(* IEC 61131-3 sources: programs/VI-54/VI-54_20171205/VI-54_20171205/Stations/Screen/LseClass170718/Class/SleegersControl, 1 file *)

(* ---- SleegersControl.st ---- *)
(*!
<Class
	Name               = "SleegersControl"
	Revision           = "0.0"
	RealtimeTask       = "false"
	CyclicTask         = "true"
	BackgroundTask     = "false"
	Sigmatek           = "false"
	OSInterface        = "false"
	HighPriority       = "false"
	Automatic          = "false"
	UpdateMode         = "Prescan"
	SharedCommandTable = "true"
	Objectsize         = "(570,120)">
	<Channels>
		<Server Name="BackToOldScreen" Visualized="true" Initialize="false" WriteProtected="false" Retentive="false"/>
		<Server Name="CarButtonHw" Visualized="true" Initialize="false" WriteProtected="true" Retentive="false"/>
		<Server Name="CarRecipes" Visualized="true" Initialize="false" WriteProtected="false" Retentive="false"/>
		<Server Name="ClassSvr" Visualized="false" Initialize="false" WriteProtected="true" Retentive="false"/>
		<Server Name="Index" Visualized="true" Initialize="false" WriteProtected="false" Retentive="false"/>
		<Server Name="OffsetCaroucelHw" Visualized="true" Initialize="false" WriteProtected="false" Retentive="false"/>
		<Server Name="ScrollBar" Visualized="true" Initialize="false" WriteProtected="false" Retentive="false"/>
		<Client Name="coAccessControlMain" Required="true" Internal="false"/>
		<Client Name="CommTerminal" Required="true" Internal="false"/>
		<Client Name="NewScreen" Required="true" Internal="false"/>
	</Channels>
</Class>
*)
SleegersControl : CLASS
  //Servers:
	ClassSvr 	: SvrChCmd_DINT;
	OffsetCaroucelHw 	: SvrCh_DINT;
	CarButtonHw 	: SvrCh_DINT;
	CarRecipes 	: SvrCh_DINT;
	Index 	: SvrCh_DINT;
	BackToOldScreen 	: SvrCh_DINT;
	ScrollBar 	: SvrCh_DINT;
  //Clients:
	coAccessControlMain 	: CltChCmd_AccessControlMain;
	NewScreen 	: CltCh_DINT;
	CommTerminal 	: CltChCmd_TerminalControl;
  //Variables:
		OldScreenNbr 	: DINT;
		Offset 	: DINT;
		OldScreen 	: DINT;
		ActScreen 	: DINT;
  //Functions:

	FUNCTION VIRTUAL GLOBAL Init;

	FUNCTION VIRTUAL GLOBAL CyWork
		VAR_INPUT
			EAX 	: UDINT;
		END_VAR
		VAR_OUTPUT
			state (EAX) 	: UDINT;
		END_VAR;

	FUNCTION GLOBAL OpenScreenAfterUnlock;

	FUNCTION VIRTUAL GLOBAL OffsetCaroucelHw::Write
		VAR_INPUT
			input (EAX) 	: DINT;
		END_VAR
		VAR_OUTPUT
			result (EAX) 	: DINT;
		END_VAR;

	FUNCTION VIRTUAL GLOBAL CarRecipes::Write
		VAR_INPUT
			input (EAX) 	: DINT;
		END_VAR
		VAR_OUTPUT
			result (EAX) 	: DINT;
		END_VAR;

	FUNCTION VIRTUAL GLOBAL Index::Write
		VAR_INPUT
			input (EAX) 	: DINT;
		END_VAR
		VAR_OUTPUT
			result (EAX) 	: DINT;
		END_VAR;

	FUNCTION VIRTUAL GLOBAL BackToOldScreen::Write
		VAR_INPUT
			input (EAX) 	: DINT;
		END_VAR
		VAR_OUTPUT
			result (EAX) 	: DINT;
		END_VAR;
  //Tables:
	FUNCTION @STD
		VAR_OUTPUT
			ret_code	: CONFSTATES;
		END_VAR;
	FUNCTION GLOBAL TAB @CT_;
END_CLASS;

#pragma usingLtd AccessControlMain
#pragma usingLtd TerminalControl

FUNCTION VIRTUAL GLOBAL SleegersControl::Init

  // Set actScreen
  ActScreen := CommTerminal.ActScreenNbr;

 // Set carroucel te one
 CarButtonHw := 1;

 // define screen numbers
 #define SMainHardware 7

 #define SVI46 48
 #define SVI11 49
 #define SVI47 50
 #define SVI48 51
 #define SVI49 52
 #define SVI50 53

 #define Salarm 22

 // define carroucel distances (offsets)
 #define OHardwareCards 550
 #define OMainHardware 600
 #define OAlarm 829

END_FUNCTION

FUNCTION VIRTUAL GLOBAL SleegersControl::CyWork
	VAR_INPUT
		EAX 	: UDINT;
	END_VAR
	VAR_OUTPUT
		state (EAX) 	: UDINT;
	END_VAR

 #define Hardware 561
 #define Alarm 829

  // go after login to Screen the right screen
  if coAccessControlMain.ActLevel = 0 then
    OldScreenNbr := coAccessControlMain.ActLevel;
  end_if;

  if OldScreenNbr = 0 then
    if coAccessControlMain.ActLevel >= 1 then
      OpenScreenAfterUnlock();
      OldScreenNbr := 1;
    end_if;
  end_if;

  // save last screen
  if ActScreen <> CommTerminal.ActScreenNbr then
    OldScreen := ActScreen;
    ActScreen := CommTerminal.ActScreenNbr;
    ScrollBar := 0;
  end_if;

	state := READY;

END_FUNCTION

FUNCTION GLOBAL SleegersControl::OpenScreenAfterUnlock

  if CommTerminal.ActScreenNbr = 0 then
    NewScreen.Write(input:=1);
  end_if;
END_FUNCTION

FUNCTION VIRTUAL GLOBAL SleegersControl::OffsetCaroucelHw::Write
	VAR_INPUT
		input (EAX) 	: DINT;
	END_VAR
	VAR_OUTPUT
		result (EAX) 	: DINT;
	END_VAR

	OffsetCaroucelHw := input;

  // Remember old screen

  // Ckeck te right offset
  if CommTerminal.ActScreenNbr = SMAINHARDWARE then
    Offset := OMainHardware;
  elsif CommTerminal.ActScreenNbr = SVI46 |
        CommTerminal.ActScreenNbr = SVI11 |
        CommTerminal.ActScreenNbr = SVI47 |
        CommTerminal.ActScreenNbr = SVI48 |
        CommTerminal.ActScreenNbr = SVI49 |
        CommTerminal.ActScreenNbr = SVI50  then
         Offset := OHardwareCards;
  elsif CommTerminal.ActScreenNbr = SALARM then
    offset := OAlarm;
  end_if;

  // Make Carroucel button invisibel when Carroucel is visibble
  if input = 0 then
    CarButtonHw := 1;
  elsif input <= 0 & input >= (0 - (1 * Offset + 50)) then
    CarButtonHw := 2;
  elsif input <= (0 - (1 * Offset - 50)) & input >=  (0 - (2 * Offset + 50 )) then
    CarButtonHw := 3;
  elsif input <= (0 - (2 * Offset - 50)) & input >=  (0 - (3 * Offset + 50 )) then
    CarButtonHw := 4;
  elsif input <= (0 - (3 * Offset - 50)) & input >=  (0 - (4 * Offset + 50 )) then
    CarButtonHw := 5;
  elsif input <= (0 - (4 * Offset - 50)) & input >=  (0 - (5 * Offset + 50 )) then
    CarButtonHw := 6;
  end_if;

	result := OffsetCaroucelHw;

END_FUNCTION

FUNCTION VIRTUAL GLOBAL SleegersControl::CarRecipes::Write
	VAR_INPUT
		input (EAX) 	: DINT;
	END_VAR
	VAR_OUTPUT
		result (EAX) 	: DINT;
	END_VAR

	CarRecipes := input;
	result := CarRecipes;

END_FUNCTION

FUNCTION VIRTUAL GLOBAL SleegersControl::Index::Write
	VAR_INPUT
		input (EAX) 	: DINT;
	END_VAR
	VAR_OUTPUT
		result (EAX) 	: DINT;
	END_VAR

	Index := input;
	result := Index;

END_FUNCTION

FUNCTION VIRTUAL GLOBAL SleegersControl::BackToOldScreen::Write
	VAR_INPUT
		input (EAX) 	: DINT;
	END_VAR
	VAR_OUTPUT
		result (EAX) 	: DINT;
	END_VAR

	BackToOldScreen := input;

  NewScreen.Write(input:= OldScreen);

	result := BackToOldScreen;

END_FUNCTION
